PROGRAM HoldingBitCtrl
VAR
	ARfbStnDoorOpenBit : 	ARRAY [1..iStnQty] OF HoldingBitSV;
	ARfbStnDoorCloseBit : 	ARRAY [1..iStnQty] OF HoldingBitSV;

	LdDoorOpenBit: HoldingBitSV;
	LdDoorCloseBit: HoldingBitSV;

	UldDoorOpenBit: HoldingBitSV;
	UldDoorCloseBit: HoldingBitSV;

	ARfbStnDoorClampBit 			: ARRAY [1..iStnQty] OF HoldingBitSV;
	ARfbStnDoorUnclampBit 		: ARRAY [1..iStnQty] OF HoldingBitSV;

	ARfbStnCylinderFrontBit		: ARRAY [1..iStnQty] OF HoldingBitSV;
	ARfbStnCylinderBackBit		: ARRAY [1..iStnQty] OF HoldingBitSV;

	LdConveyorIn : HoldingBitSV;
	LdConveyorOut: HoldingBitSV;

	UldConveyorOpen: HoldingBitSV;
	UldConveyorClose: HoldingBitSV;

	LdConveyorUp: HoldingBitSV;
	LdConveyorDown: HoldingBitSV;

	UldConveyorUp: HoldingBitSV;
	UldConveyorDown: HoldingBitSV;

	NIL: BOOL;

END_VAR

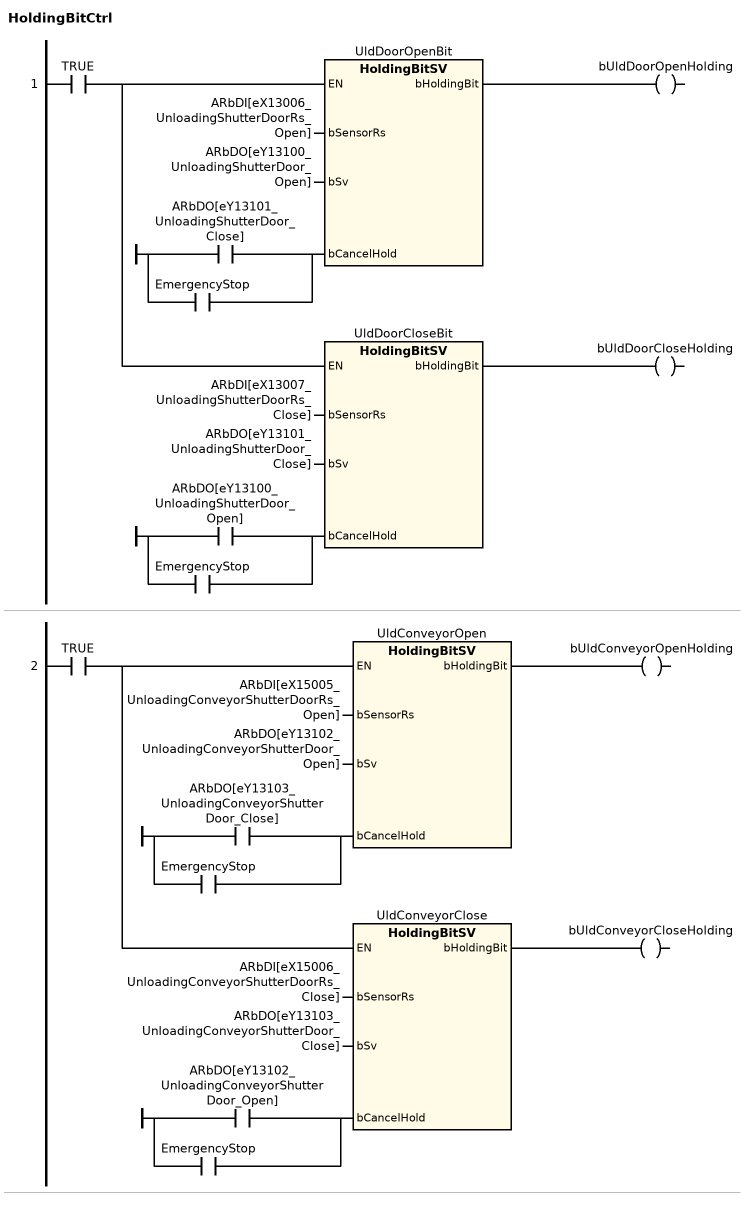
// NETWORK 1
UldDoorOpenBit(
    bSensorRs := ARbDI[eX13006_UnloadingShutterDoorRs_Open],
    bSv := ARbDO[eY13100_UnloadingShutterDoor_Open],
    bCancelHold := ARbDO[eY13101_UnloadingShutterDoor_Close] OR EmergencyStop); // HoldingBitSV
bUldDoorOpenHolding := UldDoorOpenBit.bHoldingBit;
UldDoorCloseBit(
    bSensorRs := ARbDI[eX13007_UnloadingShutterDoorRs_Close],
    bSv := ARbDO[eY13101_UnloadingShutterDoor_Close],
    bCancelHold := ARbDO[eY13100_UnloadingShutterDoor_Open] OR EmergencyStop); // HoldingBitSV
bUldDoorCloseHolding := UldDoorCloseBit.bHoldingBit;

// NETWORK 2
UldConveyorOpen(
    bSensorRs := ARbDI[eX15005_UnloadingConveyorShutterDoorRs_Open],
    bSv := ARbDO[eY13102_UnloadingConveyorShutterDoor_Open],
    bCancelHold := ARbDO[eY13103_UnloadingConveyorShutterDoor_Close] OR EmergencyStop); // HoldingBitSV
bUldConveyorOpenHolding := UldConveyorOpen.bHoldingBit;
UldConveyorClose(
    bSensorRs := ARbDI[eX15006_UnloadingConveyorShutterDoorRs_Close],
    bSv := ARbDO[eY13103_UnloadingConveyorShutterDoor_Close],
    bCancelHold := ARbDO[eY13102_UnloadingConveyorShutterDoor_Open] OR EmergencyStop); // HoldingBitSV
bUldConveyorCloseHolding := UldConveyorClose.bHoldingBit;

END_PROGRAM

(* stored: Version 1.1.0.1, ProductVersion 3.1.4024.12
   POU HoldingBitCtrl: Id {aa0857fc-7eef-4ada-825f-9b5700d4b1d8}, SpecialFunc None *)
